FUNCTION_BLOCK EnO_TK_SR65_LI
VAR_INPUT
	ID: DWORD;
END_VAR
VAR_OUTPUT
	LUX: WORD;
	status: BOOL; (*TRUE = Low Voltage; False = Voltage OK*);
END_VAR
VAR
	READ: FB_Rec_Generic;
	POWER: DINT;
END_VAR

READ(
	str_KL6581:=enocean_buffer , 
	byNode:=1 , 
	dw_ID:=ID , 
	ar_Value=> , 
	by_Node=> , 
	by_STATE=> , 
	bReceive=> , 
	EnOceanTyp=> );

LUX:=read.ar_Value[1]*4;	
POWER:=TRUNC(read.ar_Value[3]/50);
IF power < 3  THEN
	status:=TRUE;
ELSE
	status:=FALSE;
END_IF

END_FUNCTION_BLOCK

(* stored: Version 1.1.0.1, ProductVersion 3.1.4022.18
   POU EnO_TK_SR65_LI: Id {e2430ee1-5bd9-4b54-b142-5bbcf3cc26df}, SpecialFunc None *)
